{attribute 'qualified_only'}
VAR_GLOBAL PERSISTENT
    arrRack              : ARRAY[1..GVL_Config.MAX_ROWS, 1..GVL_Config.MAX_COLUMNS] OF ST_StorageSlot;
    nTotalStoredCount    : UDINT;
    nTotalRetrievedCount : UDINT;
    sWarehouseName       : STRING := 'IntimeTec_ASRS_01';
    bRackInitialized     : BOOL;
END_VAR

VAR_GLOBAL
    bSystemAutoMode      : BOOL := FALSE;
    bEmergencyStop       : BOOL := FALSE;
    sSystemStatusMsg     : STRING(80) := 'System Ready';
    stHmiSearch          : ST_HMI_Search;
	bStartRetrieval      : BOOL;
	bRetrievalRow        : INT;
	bRetrievalCol        : INT;
END_VAR

(* stored: Version 1.1.0.1, ProductVersion 3.1.4024.16
   GVL GVL_Warehouse: Id {a1b2c3d4-e5f6-7890-abcd-ef1234567890} *)
